KUKA KRL program: wkz6_ab.src, wkz6_ab.dat

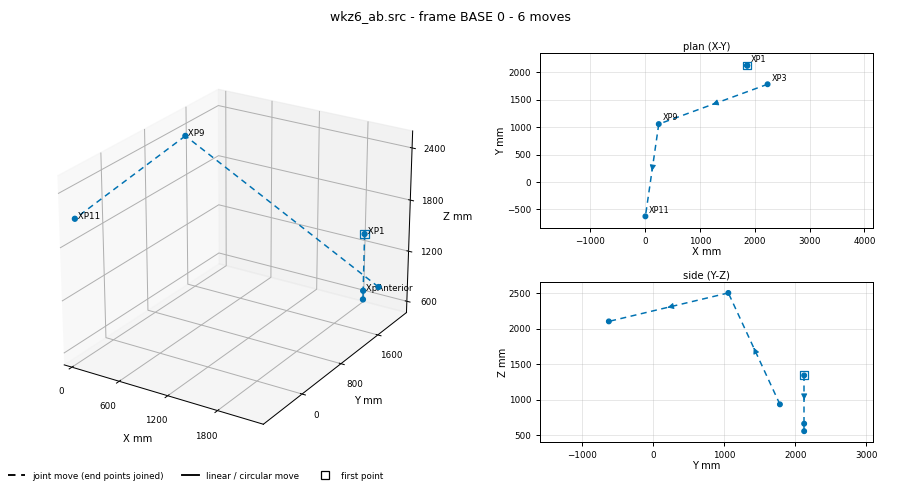
[picture p0: tool path of wkz6_ab.src in frame BASE 0, 6 of 8 moves have a stored position in this frame; points joined in program order, loops and branches not executed]
--- wkz6_ab.src ---
&ACCESS RVP2
&REL 22
&COMMENT Deposito Gripper Teto ACCELO
&PARAM DISKPATH = KRC:\R1\Program
&PARAM TEMPLATE = C:\KRC\Roboter\Template\vorgabe
&PARAM EDITMASK = *
DEF wkz6_ab( )
;FOLD INI
  ;FOLD BASISTECH INI
    GLOBAL INTERRUPT DECL 3 WHEN $STOPMESS==TRUE DO IR_STOPM ( )
    INTERRUPT ON 3
    BAS (#INITMOV,0 )
  ;ENDFOLD (BASISTECH INI)
;FOLD GRIPPERTECH INI
USER_GRP(0,DUMMY,DUMMY,GDEFAULT)
;ENDFOLD (GRIPPERTECH INI)
  ;FOLD USER INI
    ;Make your modifications here

  ;ENDFOLD (USER INI)
;ENDFOLD (INI)

; Caracterização dos meios de produção:
; Changes: Deposita Gripper Teto Accelo
; Versão Atual:13/10/2015
; Name: P13.050-R1

chk_w6_wechs_ok ( )              ; CHECK GRIPPER ACCELO

;FOLD PTP P13 CONT Vel=100 % PDAT14 Tool[8]:TOOL_CHANGER Base[2]:Accelo;%{PE}%R 8.2.20,%MKUKATPBASIS,%CMOVE,%VPTP,%P 1:PTP, 2:P13, 3:C_DIS, 5:100, 7:PDAT14
$BWDSTART=FALSE
PDAT_ACT=PPDAT14
FDAT_ACT=FP13
BAS(#PTP_PARAMS,100)
PTP XP13 C_DIS
;ENDFOLD

;FOLD WAIT FOR ( IN 219 'Posicao p/ Acoplamento OK' ) CONT;%{PE}%R 8.2.20,%MKUKATPBASIS,%CEXT_WAIT_FOR,%VEXT_WAIT_FOR,%P 2:, 4:, 5:$IN, 6:219, 7:Posicao p/ Acoplamento OK, 9:CONTINUE
CONTINUE
WAIT FOR  ( $IN[219] )
;ENDFOLD
;FOLD WAIT FOR NOT ( IN 185 'DOCK 4 Deposito Ocupado' ) CONT;%{PE}%R 8.2.20,%MKUKATPBASIS,%CEXT_WAIT_FOR,%VEXT_WAIT_FOR,%P 2:NOT, 4:, 5:$IN, 6:185, 7:DOCK 4 Deposito Ocupado, 9:CONTINUE
CONTINUE
WAIT FOR  NOT ( $IN[185] )
;ENDFOLD
;FOLD WAIT FOR ( IN 189 'DOCK 4 Proteção Aberta' ) CONT;%{PE}%R 8.2.20,%MKUKATPBASIS,%CEXT_WAIT_FOR,%VEXT_WAIT_FOR,%P 2:, 4:, 5:$IN, 6:189, 7:DOCK 4 Proteção Aberta, 9:CONTINUE
CONTINUE
WAIT FOR  ( $IN[189] )
;ENDFOLD
;FOLD WAIT FOR NOT ( IN 190 'DOCK 4 Proteção Fechada' ) CONT;%{PE}%R 8.2.20,%MKUKATPBASIS,%CEXT_WAIT_FOR,%VEXT_WAIT_FOR,%P 2:NOT, 4:, 5:$IN, 6:190, 7:DOCK 4 Proteção Fechada, 9:CONTINUE
CONTINUE
WAIT FOR  NOT ( $IN[190] )
;ENDFOLD

;FOLD PTP P1 CONT Vel=100 % PDAT1 Tool[8]:TOOL_CHANGER Base[2]:Accelo;%{PE}%R 8.2.20,%MKUKATPBASIS,%CMOVE,%VPTP,%P 1:PTP, 2:P1, 3:C_DIS, 5:100, 7:PDAT1
$BWDSTART=FALSE
PDAT_ACT=PPDAT1
FDAT_ACT=FP1
BAS(#PTP_PARAMS,100)
PTP XP1 C_DIS
;ENDFOLD
;FOLD PTP pAnterior CONT Vel=100 % PDAT7 Tool[8]:TOOL_CHANGER Base[2]:Accelo;%{PE}%R 8.2.20,%MKUKATPBASIS,%CMOVE,%VPTP,%P 1:PTP, 2:pAnterior, 3:C_DIS, 5:100, 7:PDAT7
$BWDSTART=FALSE
PDAT_ACT=PPDAT7
FDAT_ACT=FpAnterior
BAS(#PTP_PARAMS,100)
PTP XpAnterior C_DIS
;ENDFOLD

;FOLD ; PONTO DE DEPOSITO DO GRIPPER;%{PE}%R 8.2.20,%MKUKATPBASIS,%CCOMMENT,%VNORMAL,%P 2:PONTO  DE  DEPOSITO  DO  GRIPPER
;ENDFOLD
;FOLD LIN pPonto_de_entrega Vel=0.15 m/s CPDAT1 Tool[6]:GRIPPER TETO ACCELO Base[0];%{PE}%R 8.2.20,%MKUKATPBASIS,%CMOVE,%VLIN,%P 1:LIN, 2:pPonto_de_entrega, 3:, 5:0.15, 7:CPDAT1
$BWDSTART=FALSE
LDAT_ACT=LCPDAT1
FDAT_ACT=FpPonto_de_entrega
BAS(#CP_PARAMS,0.15)
LIN XpPonto_de_entrega
;ENDFOLD

;FOLD WAIT FOR ( IN 222 'Liberacao p/ Desbloqueio' );%{PE}%R 8.2.20,%MKUKATPBASIS,%CEXT_WAIT_FOR,%VEXT_WAIT_FOR,%P 2:, 4:, 5:$IN, 6:222, 7:Liberacao p/ Desbloqueio, 9:
WAIT FOR  ( $IN[222] )
;ENDFOLD
;FOLD WAIT FOR ( IN 185 'DOCK 4 Deposito Ocupado' );%{PE}%R 8.2.20,%MKUKATPBASIS,%CEXT_WAIT_FOR,%VEXT_WAIT_FOR,%P 2:, 4:, 5:$IN, 6:185, 7:DOCK 4 Deposito Ocupado, 9:
WAIT FOR  ( $IN[185] )
;ENDFOLD
;FOLD WAIT Time=0.25 sec;%{PE}%R 8.2.20,%MKUKATPBASIS,%CWAIT,%VWAIT,%P 3:0.25
WAIT SEC 0.25
;ENDFOLD
;FOLD OUT 224 'Bloquear MPS' State=FALSE ;%{PE}%R 8.2.20,%MKUKATPBASIS,%COUT,%VOUTX,%P 2:224, 3:Bloquear MPS, 5:FALSE, 6:
$OUT[224]=FALSE
;ENDFOLD
;FOLD OUT 223 'Desbloquear MPS' State=TRUE ;%{PE}%R 8.2.20,%MKUKATPBASIS,%COUT,%VOUTX,%P 2:223, 3:Desbloquear MPS, 5:TRUE, 6:
$OUT[223]=TRUE
;ENDFOLD
;FOLD WAIT FOR ( IN 217 'MPS Destravado' );%{PE}%R 8.2.20,%MKUKATPBASIS,%CEXT_WAIT_FOR,%VEXT_WAIT_FOR,%P 2:, 4:, 5:$IN, 6:217, 7:MPS Destravado, 9:
WAIT FOR  ( $IN[217] )
;ENDFOLD
;FOLD WAIT FOR NOT ( IN 221 'MPS Travado' );%{PE}%R 8.2.20,%MKUKATPBASIS,%CEXT_WAIT_FOR,%VEXT_WAIT_FOR,%P 2:NOT, 4:, 5:$IN, 6:221, 7:MPS Travado, 9:
WAIT FOR  NOT ( $IN[221] )
;ENDFOLD
;FOLD IBUS OFF;%{PE}%R 8.2.20,%MKUKATPBASIS,%CIBUS,%VMAP,%P 2:#OFF, 3:2
$IBUS_OFF=$IBUS_ON
$IBUS_ON=0
;ENDFOLD
;FOLD WAIT Time=0.5 sec;%{PE}%R 8.2.20,%MKUKATPBASIS,%CWAIT,%VWAIT,%P 3:0.5
WAIT SEC 0.5
;ENDFOLD

;FOLD LIN P2 CONT Vel=0.25 m/s CPDAT3 Tool[8]:TOOL_CHANGER Base[2]:Accelo;%{PE}%R 8.2.20,%MKUKATPBASIS,%CMOVE,%VLIN,%P 1:LIN, 2:P2, 3:C_DIS C_DIS, 5:0.25, 7:CPDAT3
$BWDSTART=FALSE
LDAT_ACT=LCPDAT3
FDAT_ACT=FP2
BAS(#CP_PARAMS,0.25)
LIN XP2 C_DIS C_DIS
;ENDFOLD

;FOLD PTP P3 CONT Vel=100 % PDAT3 Tool[8]:TOOL_CHANGER Base[2]:Accelo;%{PE}%R 8.2.20,%MKUKATPBASIS,%CMOVE,%VPTP,%P 1:PTP, 2:P3, 3:C_DIS, 5:100, 7:PDAT3
$BWDSTART=FALSE
PDAT_ACT=PPDAT3
FDAT_ACT=FP3
BAS(#PTP_PARAMS,100)
PTP XP3 C_DIS
;ENDFOLD
;FOLD PTP P9 CONT Vel=100 % PDAT10 Tool[8]:TOOL_CHANGER Base[2]:Accelo;%{PE}%R 8.2.20,%MKUKATPBASIS,%CMOVE,%VPTP,%P 1:PTP, 2:P9, 3:C_DIS, 5:100, 7:PDAT10
$BWDSTART=FALSE
PDAT_ACT=PPDAT10
FDAT_ACT=FP9
BAS(#PTP_PARAMS,100)
PTP XP9 C_DIS
;ENDFOLD

;FOLD PULSE 215 'DK 7 Pinça C1 Protecao R' State=TRUE CONT Time=1 sec;%{PE}%R 8.2.20,%MKUKATPBASIS,%COUT,%VPULSE,%P 2:215, 3:DK 7 Pinça C1 Protecao R, 5:TRUE, 6:CONTINUE, 8:1
CONTINUE
PULSE($OUT[215], TRUE,1)
;ENDFOLD
;FOLD PULSE 192 'DK 4 GRP Accelo T Protecao V' State=TRUE Time=1 sec;%{PE}%R 8.2.20,%MKUKATPBASIS,%COUT,%VPULSE,%P 2:192, 3:DK 4 GRP Accelo T Protecao V, 5:TRUE, 6:, 8:1
PULSE($OUT[192], TRUE,1)
;ENDFOLD

;FOLD PTP P11 CONT Vel=100 % PDAT12 Tool[8]:TOOL_CHANGER Base[0];%{PE}%R 8.2.20,%MKUKATPBASIS,%CMOVE,%VPTP,%P 1:PTP, 2:P11, 3:C_DIS, 5:100, 7:PDAT12
$BWDSTART=FALSE
PDAT_ACT=PPDAT12
FDAT_ACT=FP11
BAS(#PTP_PARAMS,100)
PTP XP11 C_DIS
;ENDFOLD

END

--- wkz6_ab.dat ---
&ACCESS RVP2
&REL 22
&COMMENT Deposito Gripper Teto ACCELO
&PARAM DISKPATH = KRC:\R1\Program
&PARAM TEMPLATE = C:\KRC\Roboter\Template\vorgabe
&PARAM EDITMASK = *
DEFDAT  wkz6_ab
;FOLD EXTERNAL DECLARATIONS;%{PE}%MKUKATPBASIS,%CEXT,%VCOMMON,%P
;FOLD GRIPPERTECH EXT
EXT  H50 (INT  :IN,INT  :IN,INT  :IN,GRP_TYP  :IN )
;ENDFOLD (GRIPPERTECH EXT)
;FOLD SPOTTECH EXT
EXT  USERSPOT (S_COMMAND  :IN,SPOT_TYPE  :IN )
;ENDFOLD (SPOTTECH EXT)
;FOLD BASISTECH EXT;%{PE}%MKUKATPBASIS,%CEXT,%VEXT,%P
EXT  BAS (BAS_COMMAND  :IN,REAL  :IN )
DECL INT SUCCESS
;ENDFOLD (BASISTECH EXT)
;FOLD USER EXT;%{E}%MKUKATPUSER,%CEXT,%VEXT,%P
;Make your modifications here

;ENDFOLD (USER EXT)
;ENDFOLD (EXTERNAL DECLARATIONS)
DECL BASIS_SUGG_T LAST_BASIS={POINT1[] "P0                      ",POINT2[] "P0                      ",CP_PARAMS[] "CPDAT0                  ",PTP_PARAMS[] "PDAT0                   ",CONT[] "                        ",CP_VEL[] "0.15                    ",PTP_VEL[] "100                     ",SYNC_PARAMS[] "SYNCDAT                 ",SPL_NAME[] "S0                      "}
DECL E6POS XP1={X 1862.28601,Y 2124.21704,Z 1340.07996,A -1.86292899,B -0.583588123,C 179.636505,S 2,T 3,E1 220.4142,E2 0.0,E3 0.0,E4 0.0,E5 0.0,E6 0.0}
DECL FDAT FP1={TOOL_NO 6,BASE_NO 0,IPO_FRAME #BASE,POINT2[] " ",TQ_STATE FALSE}
DECL PDAT PPDAT1={VEL 100.0,ACC 100.0,APO_DIST 100.0,APO_MODE #CDIS}
DECL LDAT LCPDAT1={VEL 2.0,ACC 100.0,APO_DIST 100.0,APO_FAC 50.0,AXIS_VEL 100.0,AXIS_ACC 100.0,ORI_TYP #VAR,CIRC_TYP #BASE,JERK_FAC 50.0,GEAR_JERK 50.0,EXAX_IGN 0}
DECL E6POS XPANTERIOR={X 1862.28699,Y 2124.21704,Z 660.080078,A -0.0584938303,B -0.583629012,C 179.636505,S 2,T 3,E1 220.413895,E2 0.0,E3 0.0,E4 0.0,E5 0.0,E6 0.0}
DECL FDAT FpAnterior={TOOL_NO 6,BASE_NO 0,IPO_FRAME #BASE,POINT2[] " ",TQ_STATE FALSE}
DECL E6POS XP2={X 3334.21606,Y -10342.1104,Z -859.374023,A 119.9384,B -0.199997097,C -179.342194,S 2,T 3,E1 220.412903,E2 0.0,E3 0.0,E4 0.0,E5 0.0,E6 0.0}
DECL FDAT FP2={TOOL_NO 8,BASE_NO 2,IPO_FRAME #BASE,POINT2[] " ",TQ_STATE FALSE}
DECL LDAT LCPDAT3={VEL 2.0,ACC 100.0,APO_DIST 100.0,APO_FAC 50.0,AXIS_VEL 100.0,AXIS_ACC 100.0,ORI_TYP #VAR,CIRC_TYP #BASE,JERK_FAC 50.0,GEAR_JERK 50.0,EXAX_IGN 0}
DECL E6POS XP3={X 2233.81689,Y 1782.66504,Z 932.413086,A -105.0616,B -0.199996293,C -179.342194,S 2,T 3,E1 220.412598,E2 0.0,E3 0.0,E4 0.0,E5 0.0,E6 0.0}
DECL FDAT FP3={TOOL_NO 8,BASE_NO 0,IPO_FRAME #BASE,POINT2[] " ",TQ_STATE FALSE}
DECL PDAT PPDAT3={VEL 100.0,ACC 100.0,APO_DIST 100.0,APO_MODE #CDIS}
DECL E6POS XpPonto_de_entrega={X 1862.29004,Y 2124.21704,Z 554.40918,A -0.058483649,B -0.583800018,C 179.636597,S 2,T 3,E1 220.4133,E2 0.0,E3 0.0,E4 0.0,E5 0.0,E6 0.0}
DECL FDAT FpPonto_de_entrega={TOOL_NO 6,BASE_NO 0,IPO_FRAME #BASE,POINT2[] " ",TQ_STATE FALSE}
DECL PDAT PPDAT7={VEL 100.0,ACC 100.0,APO_DIST 100.0,APO_MODE #CDIS}
DECL E6POS XP9={X 249.382996,Y 1056.52698,Z 2501.11694,A -7.50005484,B -8.73288345,C -171.162506,S 2,T 3,E1 163.542999,E2 0.0,E3 0.0,E4 0.0,E5 0.0,E6 0.0}
DECL FDAT FP9={TOOL_NO 8,BASE_NO 0,IPO_FRAME #BASE,POINT2[] " ",TQ_STATE FALSE}
DECL PDAT PPDAT10={VEL 100.0,ACC 100.0,APO_DIST 100.0,APO_MODE #CDIS}
DECL E6POS XP11={X 5.94592714,Y -626.071716,Z 2100.45996,A -77.0253677,B -9.68873405,C 176.383698,S 2,T 2,E1 213.663498,E2 0.0,E3 0.0,E4 0.0,E5 0.0,E6 0.0}
DECL FDAT FP11={TOOL_NO 8,BASE_NO 0,IPO_FRAME #BASE,POINT2[] " ",TQ_STATE FALSE}
DECL PDAT PPDAT12={VEL 100.0,ACC 100.0,APO_DIST 100.0,APO_MODE #CDIS}
DECL E6POS XP13={X 3545.5979,Y -9867.09473,Z 204.327393,A -135.625198,B -17.27075,C -179.614594,S 2,T 3,E1 220.305695,E2 0.0,E3 0.0,E4 0.0,E5 0.0,E6 0.0}
DECL FDAT FP13={TOOL_NO 6,BASE_NO 2,IPO_FRAME #BASE,POINT2[] " ",TQ_STATE FALSE}
DECL PDAT PPDAT14={VEL 100.0,ACC 100.0,APO_DIST 100.0,APO_MODE #CDIS}
DECL E6POS XP4={X 3545.5979,Y -9867.09473,Z 204.327393,A -135.625198,B -17.27075,C -179.614594,S 2,T 3,E1 220.305695,E2 0.0,E3 0.0,E4 0.0,E5 0.0,E6 0.0}
DECL FDAT FP4={TOOL_NO 6,BASE_NO 2,IPO_FRAME #BASE,POINT2[] " ",TQ_STATE FALSE}
DECL PDAT PPDAT2={VEL 100.0,ACC 100.0,APO_DIST 100.0,APO_MODE #CDIS}
ENDDAT
